(* CODESYS project MOTORES_SEQUENCIA.project

Project tree, tasks and I/O mapping:
  Device : CODESYS Control Win V3, 3S - Smart Software Solutions GmbH, order no. 305021, version 3.5.11.30
    application Application
      libraries: Standard, * (System)
      task MainTask (cyclic, interval t#20ms, priority 1) calls PLC_PRG
      task VISU_TASK (cyclic, interval 100 ms, priority 31) calls VisuElems.Visu_Prg
      program PLC_PRG [LD]
      visualisation Visualization
  libraries: VisuSymbols, 3.5.10.0 (System)
  text list GlobalTextList
*)

// Device/Application/PLC_PRG
PROGRAM PLC_PRG
VAR
	CH : BOOL;
	M1 : BOOL;
	M2 : BOOL;
	TON_1: TON;
	TON_2: TON;
	T1: TIME;
	T2: TIME;
	TON_3: TON;
	TON_4: TON;
	M4: BOOL;
	M3: BOOL;
	T3: TIME;
	T4: TIME;
	M5: BOOL;
	M6: BOOL;
	M7: BOOL;
	T5: TIME;
	T6: TIME;
	T7: TIME;
	TON_5: TON;
	TON_6: TON;
	TON_7: TON;
	TOF_1: TOF;
	TF1: TIME;
	CHD: BOOL;
END_VAR

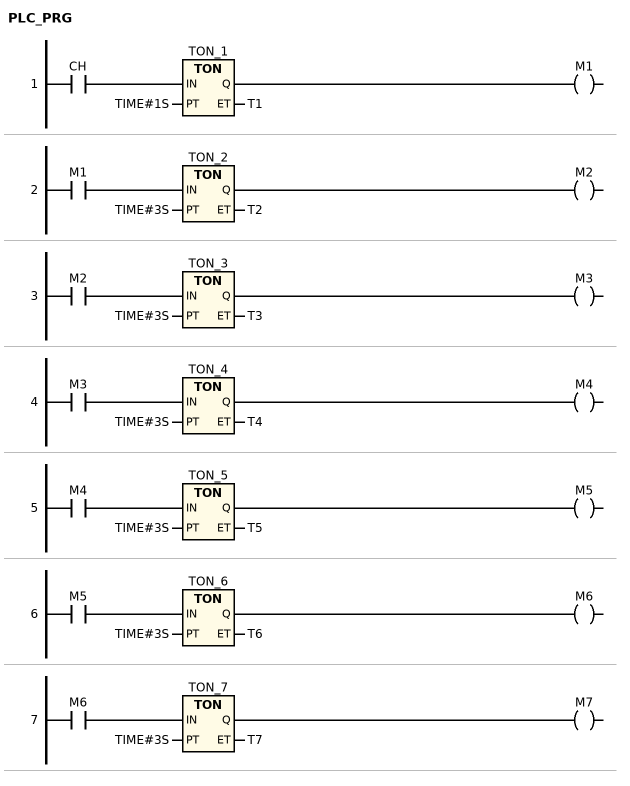
// NETWORK 1
TON_1(IN := CH, PT := TIME#1S, ET => T1); // TON
M1 := TON_1.Q;

// NETWORK 2
TON_2(IN := M1, PT := TIME#3S, ET => T2); // TON
M2 := TON_2.Q;

// NETWORK 3
TON_3(IN := M2, PT := TIME#3S, ET => T3); // TON
M3 := TON_3.Q;

// NETWORK 4
TON_4(IN := M3, PT := TIME#3S, ET => T4); // TON
M4 := TON_4.Q;

// NETWORK 5
TON_5(IN := M4, PT := TIME#3S, ET => T5); // TON
M5 := TON_5.Q;

// NETWORK 6
TON_6(IN := M5, PT := TIME#3S, ET => T6); // TON
M6 := TON_6.Q;

// NETWORK 7
TON_7(IN := M6, PT := TIME#3S, ET => T7); // TON
M7 := TON_7.Q;

END_PROGRAM

// Device/Application/Visualization
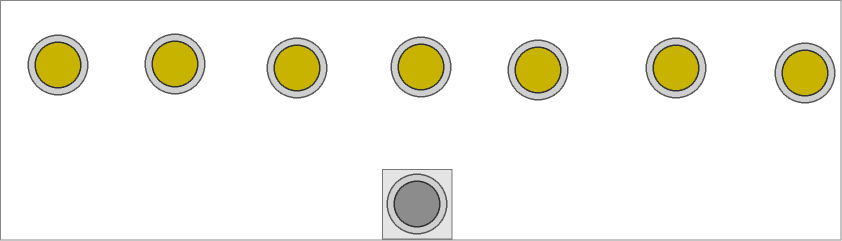
VISUALIZATION Visualization  // 842x241
    Lamp1 (23,30 70x70), variable: PLC_PRG.M1, style: Lamp-Lamp1-Yellow
    PushSwitchLed (382,169 70x70), variable: PLC_PRG.CH, behaviour: TOGGLE, style: Switch-PushSwitchLed-Gray
    Lamp1 (262,33 70x70), variable: PLC_PRG.M3, style: Lamp-Lamp1-Yellow
    Lamp1 (641,33 70x70), variable: PLC_PRG.M6, style: Lamp-Lamp1-Yellow
    Lamp1 (770,38 70x70), variable: PLC_PRG.M7, style: Lamp-Lamp1-Yellow
    Lamp1 (386,32 70x70), variable: PLC_PRG.M4, style: Lamp-Lamp1-Yellow
    Lamp1 (503,35 70x70), variable: PLC_PRG.M5, style: Lamp-Lamp1-Yellow
    Lamp1 (140,29 70x70), variable: PLC_PRG.M2, style: Lamp-Lamp1-Yellow
END_VISUALIZATION
